// TIA Portal V18 program export: 1 tag tables, 3 data types, 16 data blocks, 44 code blocks (in call order from the OBs), 85 instance data blocks

VAR_GLOBAL   // PLC tag table "Default tag table"
   ESTOP_Button AT %I0.0 : Bool;   // Emergency button
   JOGNEG_BTN_Z1 AT %I0.2 : Bool;   // Z1 - Jogging Negative -> In order to execute this, real button sholud be pressed
   JOGPOS_BTN_Z1 AT %I0.1 : Bool;   // Z1 - Jogging Positive -> In order to execute this, real button sholud be pressed
   JOGNEG_BTN_Z2 AT %I0.4 : Bool;   // Z2 - Jogging Negative -> In order to execute this, real button sholud be pressed
   JOGPOS_BTN_Z2 AT %I0.3 : Bool;   // Z2 - Jogging Positive -> In order to execute this, real button sholud be pressed
   SENSOR_DOOR AT %I0.5 : Bool;   // Door Sensor Front
   Load_Cell_Ink AT %IW66 : UInt;
   Load_Cell_Waste AT %IW64 : UInt;
   SENSOR_DOOR_2 AT %I0.6 : Bool;   // Door Sensor Front
   UV_Error_Signal AT %I0.7 : Bool;   // Error signal from UV lamp, 0-4 V error, 16-24 V ok;
   SENSOR_DOOR_3 AT %I1.0 : Bool;   // Door Sensor Side
   SENSOR_DOOR_4 AT %I1.1 : Bool;   // Door Sensor Side
   SENSOR_DOOR_5 AT %I1.2 : Bool;   // Door Sensor Fluid Supply
   SENSOR_DOOR_6 AT %I1.3 : Bool;   // Door Sensor Fluid Supply
   TemperatureSensor AT %IW116 : UInt;
   CappingSensor AT %IW118 : UInt;
   AnalogInput3 AT %IW120 : UInt;
   AnalogInput4 AT %IW122 : UInt;
   "Roller Encoder" AT %ID1000 : DWord;
   "STO-B_Output" AT %Q0.0 : Bool;   // Safty Torque Off , for CMMO [Port X3, Pin ..]and CMMP in order to release a break
   Roller_Output AT %Q0.6 : Bool;
   Heater_Output AT %Q1.0 : Bool;   // Heater: ON/OFF_PLC/3.2B; %Q1.0
   LED_1_Output AT %Q0.4 : Bool;
   LED_2_Output AT %Q0.5 : Bool;
   Heater_PWM_pulseduration AT %QW1008 : Int;   // Heater: SETPOINT_PLC/3.2C; %Q0.3
   Capping_Station_PTO AT %Q0.1 : Bool;
   Capping_Station_DIR AT %Q0.2 : Bool;
   Roller_PWM_pulseduration AT %QW1014 : Int;
   UV_CTRL_ON_OFF AT %Q0.7 : Bool;
   UV_Dimming AT %QW106 : UInt;
   Stacklight01 AT %Q50.0 : Bool;
   Stacklight02 AT %Q50.1 : Bool;
   RollerDirection AT %Q1.1 : Bool;
   Tag_1 AT %IW1000 : Hw_Hsc;
END_VAR

TYPE "DT_FML_PRM_FILE"
   STRUCT
      Control : Int;
      BitSequenceNr : Int;
      Data : Array[1..6] of Byte;
   END_STRUCT;
END_TYPE

TYPE "DT_FML_REF"
   STRUCT
      InData : Struct
         FHPP : Array[1..16] of Byte;
         FPC : Array[1..8] of Byte;
         FHPPplus : Array[1..10] of DInt;
      END_STRUCT;
      OutData : Struct
         FHPP : Array[1..16] of Byte;
         FPC : Array[1..8] of Byte;
         FHPPplus : Array[1..10] of DInt;
      END_STRUCT;
      Modbus : Bool;
      DeviceType : String[16];
      MemberID : Int;
      MemberIDmax : Int;
      Done : Bool;
      Err : Bool;
      PNU : Word;
      ActPNU : Word;
      ReqID : Int;
      RespID : Int;
      FPCC_Modus : Byte;
      FPCS_Modus : Byte;
      FPCC_Packet : "DT_FML_PRM_FILE";
      FPCS_Packet : "DT_FML_PRM_FILE";
      Subindex : Byte;
      ActSubindex : Byte;
      DatatypeWR : Byte;
      DatatypeRD : Byte;
      ParamValueWR : DInt;
      ParamValueRD : DInt;
   END_STRUCT;
END_TYPE

TYPE "DT_FML_STATUS"
   STRUCT
      Err : Bool;
      Cat : Int;
      ID : DInt;
   END_STRUCT;
END_TYPE

DATA_BLOCK "Auxiliary_variables"   // DB17
{ S7_Optimized_Access := 'TRUE' }
VERSION : 0.1
   VAR
      GlobalEnableAxis : Bool;   // Variable enables Enable_machine [FC5]
      DisableAxis : Bool;   // Variable enables Stop_machine_sequence [FC4]
      StartFunction : Bool;   // Variable enables Function_sequence [FC6]
      ESTOP : Bool;   // Variable enables Emergancy_stop_sequence [FC3]
      ResetErrors : Bool;   // Variable enables Reset_error_sequence [FB14]
      Position_range_Z2 : DInt;   // Check if position is in the range Z2
      Mov_permission_Z2_Absolute : Bool;   // Permission to move Z2 (Input Axis_Mov Z2)
      Mov_permission_Z2_Relative : Bool;
      Stop_Z2_Out : Bool;   // Stop Z2 movement (Output for Axis_Mov Z2 block)
      Reset_command_Z2 : Bool;   // Reset Mov_mode / Mode_mode = 0 / Input for BOOL_DEMUX and Output for Axis_Mov Z2 Block
      Reset_error_jump_Z2 : Bool;   // Using in order to eliminate double write
      Position_range_X : DInt;   // Check if position is in the range X
      Mov_permission_X_Absolute : Bool;   // Permission to move Z2 (Input Axis_Mov X)
      Mov_permission_X_Relative : Bool;
      Stop_X_Out : Bool;   // Stop X movement (Output for Axis_Mov X block)
      Reset_command_X : Bool;   // Reset Mov_mode / Mode_mode = 0 / Input for BOOL_DEMUX and Output for Axis_Mov X Block
      Reset_error_jump_X : Bool;   // Using in order to eliminate double write
      Reset_command_Y : Bool;   // Reset Mov_mode / Mode_mode = 0 / Input for BOOL_DEMUX and Output for Axis_Mov Y Block
      Reset_error_jump_Y : Bool;   // Using in order to eliminate double write
      Stop_Y_Out : Bool;   // Stop Y movement (Output for Axis_Mov Y block)
      Mov_permission_Y_Absolute : Bool;   // Permission to move Y (Input Axis_Mov Y)
      Mov_permission_Y_Relative : Bool;
      Position_range_Y : DInt;   // Check if position is in the range Y
      Position_range_Z1 : DInt;   // Check if position is in the range Z1
      Mov_permission_Z1_Absolute : Bool;   // Permission to move Z1 (Input Axis_Mov Z1)
      Mov_permission_Z1_Relative : Bool;
      Stop_Z1_Out : Bool;   // Stop Z1 movement (Output for Axis_Mov Z1 block)
      Reset_command_Z1 : Bool;   // Reset Mov_mode / Mode_mode = 0 / Input for BOOL_DEMUX and Output for Axis_Mov Z1 Block
      Reset_error_jump_Z1 : Bool;   // Using in order to eliminate double write
      Stop_all_axis_command : Bool;   // Execute via Step6 ( in Main) / Stop all axis
      Mov_mode_reset_ALL_Axis : Bool;   // Reset Mov_mode after stopping all axis
      JogPosBTN_Z1_RisingEdge : Bool;   // Auxiliary variable used to execute JogPos Button
      JogNegBTN_Z1_RisingEdge : Bool;   // Auxiliary variable used to execute JogNeg Button
      JogPosBTN_Z1_FallingEdge : Bool;   // Auxiliary variable used to execute JogPos Button
      JogNegBTN_Z1_FallingEdge : Bool;   // Auxiliary variable used to execute JogNeg Button
      JogPosBTN_Z2_RisingEdge : Bool;   // Auxiliary variable used to execute JogPos Button
      JogNegBTN_Z2_RisingEdge : Bool;   // Auxiliary variable used to execute JogNeg Button
      JogPosBTN_Z2_FallingEdge : Bool;   // Auxiliary variable used to execute JogPos Button
      JogNegBTN_Z2_FallingEdge : Bool;   // Auxiliary variable used to execute JogNeg Button
      Heater_Start : Bool;   // Variable used to activate the heater during the spreading sequence
      PID_PWM_Output : Bool;   // PID Compact block -> Output
      CMD_Y_EM : Bool;
      CMD_X_EM : Bool;
      CMD_Z1_EM : Bool;
      CMD_Z2_EM : Bool;
      RelativeZ1 : Bool;
   END_VAR
BEGIN
END_DATA_BLOCK

DATA_BLOCK "ChaosDB"   // DB18
{ S7_Optimized_Access := 'TRUE' }
VERSION : 0.1
   VAR
      Step0 : Bool;
      Step1 : Bool;
      Step2 : Bool;
      Step3 : Bool;
      Step4 : Bool;
      Step5 : Bool;
      Step6 : Bool;
      Step7 : Bool;
      Step10 : Bool;
      Step20 : Bool;
      Step21 : Bool;
      Step1_Step2 : Bool;
      Step2_Step3 : Bool;
      Step2_Step5 : Bool;
      Step4_Step5 : Bool;
      Step2_Step20 : Bool;
      Step3_Step_4 : Bool;
      Step4_Step6 : Bool;
      Step4_Step10 : Bool;
      Step4_Step20 : Bool;
      Step5_Step2 : Bool;
      Step6_Step7 : Bool;
      Step7_Step4 : Bool;
      Step10_Step2 : Bool;
      Step20_Step21 : Bool;
      Step21_Step2 : Bool;
      Edge_Step1M : Bool;
      Edge_Step1S : Bool;
      Edge_Reset_Z2_M : Bool;
      Edge_Reset_Z2_S : Bool;
      Edge_Reset_X_S : Bool;
      Edge_Reset_X_M : Bool;
      Edge_Reset_Y_S : Bool;
      Edge_Reset_Y_M : Bool;
      Reset_error_main : Bool;
      Edge_M_res_err_main : Bool;
      Edge_S_res_err_main : Bool;
      Edge_Reset_Z1_S : Bool;
      Edge_Reset_Z1_M : Bool;
      Monitor_state : Bool;   // Auxiliary variable
      Edge_S_ResCMMOZ2 : Bool;   // Reset CMMO Z2 Controller
      Edge_M_ResCMMOZ2 : Bool;   // Reset CMMO Z2 Controller
      Restart_CMMO_Z2_Cmd : Bool;   // Reset CMMO Z2 Controller
      Edge_S_ResCMMOZ1 : Bool;   // Reset CMMO Z1Controller
      Edge_M_ResCMMOZ1 : Bool;   // Reset CMMO Z1 Controller
      Restart_CMMO_Z1_Cmd : Bool;   // Reset CMMO Z1Controller
      Edge_S_ResCMMPX : Bool;   // Reset CMMP X Controller
      Edge_M_ResCMMPX : Bool;   // Reset CMMP X Controller
      Restart_CMMP_X_Cmd : Bool;   // Reset CMMP X Controller
      Edge_S_ResCMMPY : Bool;   // Reset CMMP Y Controller
      Edge_M_ResCMMPY : Bool;   // Reset CMMP Y Controller
      Restart_CMMP_Y_Cmd : Bool;   // Reset CMMP Y Controller
      Z2_Stop_E : Bool;
      Z2_Stop_EM : Bool;
   END_VAR
BEGIN
END_DATA_BLOCK

DATA_BLOCK "DevTestBlock"   // DB47
{ S7_Optimized_Access := 'FALSE' }
VERSION : 0.1
   VAR
      EnableAxisTest : Bool;
      Z2Halt : Bool;
      Z1Halt : Bool;
      XHalt : Bool;
      YHalt : Bool;
      GlobalHalt : Bool;
      TaskZ2E : Bool;
      TaskZ1M : Bool;
      TaskZ2M : Bool;
      TaskXM : Bool;
      TaskYM : Bool;
      TestResetCommand : Bool;
      TestResetZ1 : Bool;
      TestResetZ2 : Bool;
      TestResetX : Bool;
      TestResetY : Bool;
      DoorSensor : Bool := true;   // True for testing to disable door sensors
      "Weight Test value" : UInt;
      DoorSensorPrintboxSkip : Bool := true;
      DoorSensor_Side : Bool := false;
      DoorSensor_PrintBox : Bool;
      AXIS_ackerror : Bool;
      AXIS_X_enable : Bool;
      AXIS_Y_enable : Bool;
      AXIS_Z1_enable : Bool;
      AXIS_jog1 : Bool := false;
      AXIS_jog2 : Bool;
      AXIS_X_velocity : Real;
      AXIS_X_position : Int;
      AXIS_execute : Bool;
      ConfigEPos : DWord := 16#0000_000F;
      "AXIS Warning" : Bool := false;
      "AXIS Error Fault" : Bool := false;
      "AXIS Enabled" : Bool := false;
      "AXIS Ready" : Bool := false;
      PurgeX : DInt := 480000;
      PurgeY : DInt := 90000;
      PurgeVelocity : DInt := 300;
      PurgeMove : Bool;
      "OLD off" : Bool;
      LED1 : Bool;
      LED2 : Bool;
      CappingHoming : Bool;
      reset : Bool;
      DamagedDoorSensorTemp : Bool := false;
      CappingEnable : Bool;
      TestYvelocity : DInt := 100000;
      TestingCappingStation : Bool;
      TestCapping01 : Bool;
      TestCapping02 : Bool;
      TestCapping03 : Bool;
      TestCappingNotUsed : Bool;
      ResetCounters : Bool;
      RET_VAL : Int;
      WebServerTest : Int := 1;
   END_VAR
BEGIN
END_DATA_BLOCK

DATA_BLOCK "MachineDB"   // DB22
{ S7_Optimized_Access := 'FALSE' }
VERSION : 0.1
   VAR RETAIN
      SerialNumber : Int := 2011;
      AutomateVersion : Int := 6;
      MachineType : String := 'ArmadilloV7BR';   // Not writable from HMI
      MachineLimit : Struct
         XSafety : Struct
            PosMax : DInt := 0;
            PosMin : DInt := 0;
            SafetyMargin : DInt;
            VelocityMax : DInt;
            VelocityMin : DInt;
         END_STRUCT;
         YSafety : Struct
            PosMax : DInt := 0;
            PosMin : DInt := 0;
            SafetyMargin : DInt;
            VelocityMax : DInt;
            VelocityMin : DInt;
         END_STRUCT;
         Z1Safety : Struct
            PosMax : DInt := 0;
            PosMin : DInt := 0;
            SafetyMargin : DInt;
            VelocityMax : DInt;
            VelocityMin : DInt;
         END_STRUCT;
         Z2Safety : Struct
            PosMax : DInt := 0;
            PosMin : DInt := 0;
            SafetyMargin : DInt;
            VelocityMax : DInt;
            VelocityMin : DInt;
         END_STRUCT;
         Heater : Struct
            FeedboxStart : DInt;
            FeedboxEnd : DInt;
            PrintboxStart : DInt;
            PrintboxEnd : DInt;
         END_STRUCT;
      END_STRUCT;
      ArmadilloOption : Struct
         MachineTypeNext : String := 'ArmadilloV7BR';
         DoorOption : Int := 3;   // SAFETY OPTION, ASK BEFORE CHANGING
         DoorOptionNext : Int := 3;
         DepowderingBox : Int;   // 0 if no box; 1 is we use V1 of the box;
         DepowderingBoxNext : Int;   // 0 if no box; 1 is we use V1 of the box;
         ZAxisDriveOption : String := 'CMMT';   // CMMT;CMMS;
         ZAxisDriveOptionNext : String := 'CMMT';   // CMMT;CMMS;
         UVOption : Int := 1;   // 0 means no UV lamp; 1 version of the UV lamp;
         UVOptionNext : Int := 1;   // 0 means no UV lamp; 1 version of the UV lamp;
         StacklightOption : Int := 1;   // 0 means no Stacklight; 1 version of the Stacklight;
         StacklightOptionNext : Int := 1;   // 0 means no Stacklight; 1 version of the Stacklight;
         CappingStationOption : Int := 1;   // 0 means no Capping Station; 1 version of the Capping Station;
         CappingStationOptionNext : Int := 1;   // 0 means no Capping Station; 1 version of the Capping Station;
      END_STRUCT;
      MachineLimitSecondary : Struct
         NoGoZone01 : Struct   // Temporary not used -> go to DepowderingBoxDimensions
            NoGoZone01_Xstart : DInt;   // Start of the No Go Zone for Depowdering Box
            NoGoZone01_Xend : DInt;   // Start of the No Go Zone for Depowdering Box
            NoGoZone01_Ystart : DInt;   // Start of the No Go Zone for Depowdering Box
            NoGoZone01_Yend : DInt;   // End of the No Go Zone for Depowdering Box
            NoGoZone01_Z1start : DInt;   // Start of the No Go Zone for Depowdering Box
            NoGoZone01_Z1end : DInt;   // End of the No Go Zone for Depowdering Box
            NoGoZone01_Z2start : DInt;   // Start of the No Go Zone for Depowdering Box
            NoGoZone01_Z2end : DInt;   // End of the No Go Zone for Depowdering Box
         END_STRUCT;
      END_STRUCT;
      MachineTypeString : Struct
         _sArmadilloDev : String := 'ArmadilloDev';   // Not writable from HMI
         _sArmadilloV2 : String := 'ArmadilloV2';   // Not writable from HMI
         _sArmadilloBRV2 : String := 'ArmadilloBRV2';   // Not writable from HMI
         _sArmadilloXLV2 : String := 'ArmadilloXLV2';   // Not writable from HMI
         _sArmadilloXLBRV2 : String := 'ArmadilloXLBRV2';   // Not writable from HMI
         _sArmadilloV6 : String := 'ArmadilloV6';   // Machine 2007;
         _sArmadilloV6BR : String := 'ArmadilloV6BR';   // Machine 2007;
         _sArmadilloV7 : String := 'ArmadilloV7';   // Machine 2009; 2011;
         _sArmadilloV7BR : String := 'ArmadilloV7BR';   // Machine 2009; 2011;
         _sArmadilloXLV7 : String := 'ArmadilloXLV7';   // Machine 2010;
         _sArmadilloXLV7BR : String := 'ArmadilloXLV7BR';   // Machine 2010;
      END_STRUCT;
      ArmadilloDevMachine : Struct   // Software limit for the Armadillo Dev machine
         XSafety : Struct
            PosMax : DInt := 454000;
            PosMin : DInt := -3000;
            SafetyMargin : DInt := 0;
            VelocityMax : DInt := 500;
            VelocityMin : DInt := 0;
         END_STRUCT;
         YSafety : Struct
            PosMax : DInt := 1100000;
            PosMin : DInt := -3000;
            SafetyMargin : DInt := 0;
            VelocityMax : DInt := 500;
            VelocityMin : DInt;
         END_STRUCT;
         Z1Safety : Struct
            PosMax : DInt := 297850;
            PosMin : DInt := -3000;
            SafetyMargin : DInt := 0;
            VelocityMax : DInt := 20;
            VelocityMin : DInt;
         END_STRUCT;
         Z2Safety : Struct
            PosMax : DInt := 297850;
            PosMin : DInt := -3000;
            SafetyMargin : DInt := 0;
            VelocityMax : DInt := 20;
            VelocityMin : DInt;
         END_STRUCT;
         Heater : Struct
            FeedboxStart : DInt := 100000;
            FeedboxEnd : DInt := 400000;
            PrintboxStart : DInt := 300000;
            PrintboxEnd : DInt := 765000;
         END_STRUCT;
      END_STRUCT;
      ArmadilloBRMachine : Struct   // Software limit for the Armadillo Dev machine
         XSafety : Struct
            PosMax : DInt := 454000;
            PosMin : DInt := -3000;
            SafetyMargin : DInt;
            VelocityMax : DInt;
            VelocityMin : DInt;
         END_STRUCT;
         YSafety : Struct
            PosMax : DInt := 1100000;
            PosMin : DInt := -3000;
            SafetyMargin : DInt;
            VelocityMax : DInt;
            VelocityMin : DInt;
         END_STRUCT;
         Z1Safety : Struct
            PosMax : DInt := 94000;   // v1 = 210500
            PosMin : DInt := -3000;
            SafetyMargin : DInt;
            VelocityMax : DInt;
            VelocityMin : DInt;
         END_STRUCT;
         Z2Safety : Struct
            PosMax : DInt := 94000;   // v1 = 210500
            PosMin : DInt := -3000;
            SafetyMargin : DInt;
            VelocityMax : DInt;
            VelocityMin : DInt;
         END_STRUCT;
         Heater : Struct
            FeedboxStart : DInt;
            FeedboxEnd : DInt;
            PrintboxStart : DInt;
            PrintboxEnd : DInt;
         END_STRUCT;
      END_STRUCT;
      ArmadilloXLMachine : Struct   // Software limit for the Armadillo Production machine
         XSafety : Struct
            PosMax : DInt := 516000;
            PosMin : DInt := -3000;
            SafetyMargin : DInt;
            VelocityMax : DInt;
            VelocityMin : DInt;
         END_STRUCT;
         YSafety : Struct
            PosMax : DInt := 1380000;
            PosMin : DInt := -3000;
            SafetyMargin : DInt;
            VelocityMax : DInt;
            VelocityMin : DInt;
         END_STRUCT;
         Z1Safety : Struct
            PosMax : DInt := 302000;
            PosMin : DInt := -500;
            SafetyMargin : DInt;
            VelocityMax : DInt;
            VelocityMin : DInt;
         END_STRUCT;
         Z2Safety : Struct
            PosMax : DInt := 302000;
            PosMin : DInt := -500;
            SafetyMargin : DInt;
            VelocityMax : DInt;
            VelocityMin : DInt;
         END_STRUCT;
         Heater : Struct
            FeedboxStart : DInt;
            FeedboxEnd : DInt;
            PrintboxStart : DInt;
            PrintboxEnd : DInt;
         END_STRUCT;
      END_STRUCT;
      ArmadilloXLBRMachine : Struct   // Software limit for the Armadillo Production machine
         XSafety : Struct
            PosMax : DInt := 516000;
            PosMin : DInt := -3000;
            SafetyMargin : DInt;
            VelocityMax : DInt;
            VelocityMin : DInt;
         END_STRUCT;
         YSafety : Struct
            PosMax : DInt := 1380000;
            PosMin : DInt := -3000;
            SafetyMargin : DInt;
            VelocityMax : DInt;
            VelocityMin : DInt;
         END_STRUCT;
         Z1Safety : Struct
            PosMax : DInt := 210500;
            PosMin : DInt := -3000;
            SafetyMargin : DInt;
            VelocityMax : DInt;
            VelocityMin : DInt;
         END_STRUCT;
         Z2Safety : Struct
            PosMax : DInt := 210500;
            PosMin : DInt := -3000;
            SafetyMargin : DInt;
            VelocityMax : DInt;
            VelocityMin : DInt;
         END_STRUCT;
         Heater : Struct
            FeedboxStart : DInt;
            FeedboxEnd : DInt;
            PrintboxStart : DInt;
            PrintboxEnd : DInt;
         END_STRUCT;
      END_STRUCT;
      ArmadilloV6Machine : Struct   // 2007 Eurostar Software limit for the Armadillo V6 machine
         XSafety : Struct
            PosMax : DInt := 500000;
            PosMin : DInt := 0;
            SafetyMargin : DInt := 5000;
            VelocityMax : DInt := 500;
            VelocityMin : DInt := 0;
         END_STRUCT;
         YSafety : Struct
            PosMax : DInt := 1365000;
            PosMin : DInt := 0;
            SafetyMargin : DInt := 5000;
            VelocityMax : DInt := 500;
            VelocityMin : DInt;
         END_STRUCT;
         Z1Safety : Struct
            PosMax : DInt := 300000;
            PosMin : DInt := 0;
            SafetyMargin : DInt := 2000;
            VelocityMax : DInt;
            VelocityMin : DInt;
         END_STRUCT;
         Z2Safety : Struct
            PosMax : DInt := 300000;
            PosMin : DInt := 0;
            SafetyMargin : DInt := 2000;
            VelocityMax : DInt;
            VelocityMin : DInt;
         END_STRUCT;
         Heater : Struct
            FeedboxStart : DInt := 270000;
            FeedboxEnd : DInt := 580000;
            PrintboxStart : DInt := 580000;
            PrintboxEnd : DInt := 880000;
         END_STRUCT;
      END_STRUCT;
      ArmadilloV6BRMachine : Struct   // 2007 Eurostar Software limit for the Armadillo V6 Bed Reduction machine
         XSafety : Struct
            PosMax : DInt := 500000;
            PosMin : DInt := 0;
            SafetyMargin : DInt := 5000;
            VelocityMax : DInt := 500;
            VelocityMin : DInt;
         END_STRUCT;
         YSafety : Struct
            PosMax : DInt := 1365000;
            PosMin : DInt := 0;
            SafetyMargin : DInt := 5000;
            VelocityMax : DInt := 500;
            VelocityMin : DInt;
         END_STRUCT;
         Z1Safety : Struct
            PosMax : DInt := 90000;   // v1 = 210500
            PosMin : DInt := 0;
            SafetyMargin : DInt := 2000;
            VelocityMax : DInt;
            VelocityMin : DInt;
         END_STRUCT;
         Z2Safety : Struct
            PosMax : DInt := 90000;   // v1 = 210500
            PosMin : DInt := 0;
            SafetyMargin : DInt := 2000;
            VelocityMax : DInt;
            VelocityMin : DInt;
         END_STRUCT;
         Heater : Struct
            FeedboxStart : DInt := 470000;
            FeedboxEnd : DInt := 580000;
            PrintboxStart : DInt := 580000;
            PrintboxEnd : DInt := 680000;
         END_STRUCT;
      END_STRUCT;
      ArmadilloV7Machine : Struct   // 2009, 2011 Normal Software limit for the Armadillo V6 machine
         XSafety : Struct
            PosMax : DInt := 435000;
            PosMin : DInt := -3000;
            SafetyMargin : DInt := 5000;
            VelocityMax : DInt := 500;
            VelocityMin : DInt := 0;
         END_STRUCT;
         YSafety : Struct
            PosMax : DInt := 1065000;
            PosMin : DInt := -3000;
            SafetyMargin : DInt := 5000;
            VelocityMax : DInt := 500;
            VelocityMin : DInt;
         END_STRUCT;
         Z1Safety : Struct
            PosMax : DInt := 312000;
            PosMin : DInt := 0;
            SafetyMargin : DInt := 2000;
            VelocityMax : DInt;
            VelocityMin : DInt;
         END_STRUCT;
         Z2Safety : Struct
            PosMax : DInt := 312000;
            PosMin : DInt := 0;
            SafetyMargin : DInt := 2000;
            VelocityMax : DInt;
            VelocityMin : DInt;
         END_STRUCT;
         Heater : Struct
            FeedboxStart : DInt := 100000;
            FeedboxEnd : DInt := 430000;
            PrintboxStart : DInt := 430000;
            PrintboxEnd : DInt := 740000;
         END_STRUCT;
      END_STRUCT;
      ArmadilloV7BRMachine : Struct   // 2009, 2011 Normal Software limit for the Armadillo V6 Bed Reduction machine
         XSafety : Struct
            PosMax : DInt := 435000;
            PosMin : DInt := -3000;
            SafetyMargin : DInt := 5000;
            VelocityMax : DInt := 500;
            VelocityMin : DInt;
         END_STRUCT;
         YSafety : Struct
            PosMax : DInt := 1065000;
            PosMin : DInt := -3000;
            SafetyMargin : DInt := 5000;
            VelocityMax : DInt := 500;
            VelocityMin : DInt;
         END_STRUCT;
         Z1Safety : Struct
            PosMax : DInt := 86000;
            PosMin : DInt := 0;
            SafetyMargin : DInt := 2000;
            VelocityMax : DInt;
            VelocityMin : DInt;
         END_STRUCT;
         Z2Safety : Struct
            PosMax : DInt := 86000;
            PosMin : DInt := 0;
            SafetyMargin : DInt := 2000;
            VelocityMax : DInt;
            VelocityMin : DInt;
         END_STRUCT;
         Heater : Struct
            FeedboxStart : DInt := 250000;
            FeedboxEnd : DInt := 360000;
            PrintboxStart : DInt := 360000;
            PrintboxEnd : DInt := 490000;
         END_STRUCT;
      END_STRUCT;
      ArmadilloXLV7Machine : Struct   // 2010 XL Software limit for the Armadillo V6 machine
         XSafety : Struct
            PosMax : DInt := 500000;
            PosMin : DInt := -3000;
            SafetyMargin : DInt := 5000;
            VelocityMax : DInt := 500;
            VelocityMin : DInt := 0;
         END_STRUCT;
         YSafety : Struct
            PosMax : DInt := 1365000;
            PosMin : DInt := -3000;
            SafetyMargin : DInt := 5000;
            VelocityMax : DInt := 500;
            VelocityMin : DInt;
         END_STRUCT;
         Z1Safety : Struct
            PosMax : DInt := 312000;
            PosMin : DInt := 0;
            SafetyMargin : DInt := 2000;
            VelocityMax : DInt;
            VelocityMin : DInt;
         END_STRUCT;
         Z2Safety : Struct
            PosMax : DInt := 312000;
            PosMin : DInt := 0;
            SafetyMargin : DInt := 2000;
            VelocityMax : DInt;
            VelocityMin : DInt;
         END_STRUCT;
         Heater : Struct
            FeedboxStart : DInt := 150000;
            FeedboxEnd : DInt := 610000;
            PrintboxStart : DInt := 610000;
            PrintboxEnd : DInt := 1100000;
         END_STRUCT;
      END_STRUCT;
      ArmadilloXLV7BRMachine : Struct   // 2010 XL Software limit for the Armadillo V6 Bed Reduction machine
         XSafety : Struct
            PosMax : DInt := 500000;
            PosMin : DInt := -3000;
            SafetyMargin : DInt := 5000;
            VelocityMax : DInt := 500;
            VelocityMin : DInt;
         END_STRUCT;
         YSafety : Struct
            PosMax : DInt := 1365000;
            PosMin : DInt := -3000;
            SafetyMargin : DInt := 5000;
            VelocityMax : DInt := 500;
            VelocityMin : DInt;
         END_STRUCT;
         Z1Safety : Struct
            PosMax : DInt := 86000;
            PosMin : DInt := 0;
            SafetyMargin : DInt := 2000;
            VelocityMax : DInt;
            VelocityMin : DInt;
         END_STRUCT;
         Z2Safety : Struct
            PosMax : DInt := 86000;
            PosMin : DInt := 0;
            SafetyMargin : DInt := 2000;
            VelocityMax : DInt;
            VelocityMin : DInt;
         END_STRUCT;
         Heater : Struct
            FeedboxStart : DInt := 440000;
            FeedboxEnd : DInt := 620000;
            PrintboxStart : DInt := 620000;
            PrintboxEnd : DInt := 770000;
         END_STRUCT;
      END_STRUCT;
      DepowderingBoxDimensions : Struct   // Should be integrated with machine limits in the future
         DepowderingBoxHeight : DInt := 27000;
         DepowderingBoxWidth : DInt := 0;
         DepowderingBoxMargin : DInt := 3000;
         DepowderingBoxNormal : Struct
            DepowderingBoxNormalXstart : DInt := 0;
            DepowderingBoxNormalXend : DInt := 550000;
            DepowderingBoxNormalYstart : DInt := 180000;
            DepowderingBoxNormalYend : DInt := 1500000;
         END_STRUCT;
         DepowderingBoxXL : Struct
            DepowderingBoxXLXstart : DInt := 0;
            DepowderingBoxXLXend : DInt := 550000;
            DepowderingBoxXLYstart : DInt := 190000;
            DepowderingBoxXLYend : DInt := 1500000;
         END_STRUCT;
      END_STRUCT;
   END_VAR
BEGIN
END_DATA_BLOCK

DATA_BLOCK "MainDB"   // DB30
{ S7_Optimized_Access := 'TRUE' }
VERSION : 0.1
   VAR
      Monitor : Bool;
      Step0M : Bool;
      Step0 : Bool;
      Step10 : Bool;
      Step20 : Bool;
      Step30 : Bool;
      Step40 : Bool;
      Step50 : Bool;
      Step0_10 : Bool;
      Step10_20 : Bool;
      Step20_30 : Bool;
      Step30_40 : Bool;
      Step40_50 : Bool;
      Step50_10 : Bool;
      ESTOPEdgeMemory : Bool;
      ESTOPEdge : Bool;
      AllAxisFaultRelease : Bool;
      Step0MConfig : Bool;
   END_VAR
BEGIN
END_DATA_BLOCK

DATA_BLOCK "WebDB"   // DB5
{ S7_Optimized_Access := 'FALSE' }
VERSION : 0.1
   VAR
      Enabled_Devices : Bool;   // Diagnostic value, necessary in step 3 (Check if system is ready); TRUE if OK;
      Ready_Devices : Bool;   // Diagnostic value, necessary in step 3 (Check if system is ready); TRUE if OK;
      Warning_Devices : Bool;   // Diagnostic value, necessary in step 3 (Check if system is ready); TRUE if OK;
      Fault_Devices : Bool;   // Diagnostic value, necessary in step 3 (Check if system is ready); TRUE if OK;
      diagMode : UInt := 1;   // Diagnostic mode : 0
      myLADDR : HW_ANY := 52;   // ID of CPUExecutUnit : 52 PLC ID: 64
      returnValue : Int;   // No error: 0
      CountDiagDetails : UInt;   // Should always be 0
      PLCDiag : DIS;   // Read value of diagnostic
      Start_Machine : Bool;   // Button - Start Machine
      Stop_Machine : Bool;   // Button - Stop Machine
      Reset_error : Bool;   // Button - Reset error after emergancy stop and other situation
      Stop_All_Axis : Bool;
      XInput : Struct
         EnableDrive : Bool;
         Stop : Bool;
         Halt : Bool;
         Brake : Bool;
         ResetFault : Bool;
         HMIAccessLocked : Bool;
         OPM : Int;   // Operating Mode ???
         StartTask : Bool;
         StartHoming : Bool;
         JogPos : Bool;
         JogNeg : Bool;
         TeachActValue : Bool;
         ClearRemPos : Bool;
         Relative : Bool;
         DeactivateStrokeLimit : Bool;
         ExecuteFunction : Bool;
         RecordNo : Int;
         SetFunctionNumber : Int;
         SetFunctionGroup : Int;
         SetValueVelocity : DInt := 20;
         SetValuePosition : DInt;
         SetValueForceRamp : DInt;
         SetValueForce : DInt;
         SetValueRotRamp : DInt;
         SetValueRotSpeed : DInt;
      END_STRUCT;
      XOutput : Struct
         DriveEnabled : Bool;
         Ready : Bool;
         Warning : Bool;
         Fault : Bool;
         SupplyVoltPresent : Bool;
         ControlFCT_HMI : Bool;
         StateOPM : Int;
         HaltNotActive : Bool;
         AckStart : Bool;
         MC : Bool;
         AckTeach : Bool;
         DriveMoving : Bool;
         DragError : Bool;
         StandStillControl : Bool;
         HomingValid : Bool;
         ActualRecordNo : Int;
         RC1 : Bool;
         RCC : Bool;
         VelocityLimitReached : Bool;
         StrokeLimitReached : Bool;
         FunctionIsActive : Bool;
         ActualFunctionNumber : Int;
         ActualFunctionGroup : Int;
         ActualPosition : DInt;
         ActualVelocity : DInt;
         ActualForce : DInt;
         ActualRotRamp : DInt;
         ActualRotSpeed : DInt;
      END_STRUCT;
      XAddOn1 : Struct
         XTargetRange : DInt := 1000;
         XTargetReached : Bool;
         XOverrange : Bool;
         Error_message_X : DInt;   // Number of error in DINT. Check error in CMMP documentation
         Restart_CMMO_X : Bool;   // Restart CMMP X controller
      END_STRUCT;
      YInput : Struct
         EnableDrive : Bool;
         Stop : Bool;
         Halt : Bool;
         Brake : Bool;
         ResetFault : Bool;
         HMIAccessLocked : Bool;
         OPM : Int;   // Operating Mode ???
         StartTask : Bool;
         StartHoming : Bool;
         JogPos : Bool;
         JogNeg : Bool;
         TeachActValue : Bool;
         ClearRemPos : Bool;
         Relative : Bool;
         DeactivateStrokeLimit : Bool;
         ExecuteFunction : Bool;
         RecordNo : Int;
         SetFunctionNumber : Int;
         SetFunctionGroup : Int;
         SetValueVelocity : DInt := 20;
         SetValuePosition : DInt;
         SetValueForceRamp : DInt;
         SetValueForce : DInt;
         SetValueRotRamp : DInt;
         SetValueRotSpeed : DInt;
      END_STRUCT;
      YOutput : Struct
         DriveEnabled : Bool;
         Ready : Bool;
         Warning : Bool;
         Fault : Bool;
         SupplyVoltPresent : Bool;
         ControlFCT_HMI : Bool;
         StateOPM : Int;
         HaltNotActive : Bool;
         AckStart : Bool;
         MC : Bool;
         AckTeach : Bool;
         DriveMoving : Bool;
         DragError : Bool;
         StandStillControl : Bool;
         HomingValid : Bool;
         ActualRecordNo : Int;
         RC1 : Bool;
         RCC : Bool;
         VelocityLimitReached : Bool;
         StrokeLimitReached : Bool;
         FunctionIsActive : Bool;
         ActualFunctionNumber : Int;
         ActualFunctionGroup : Int;
         ActualPosition : DInt;
         ActualVelocity : DInt;
         ActualForce : DInt;
         ActualRotRamp : DInt;
         ActualRotSpeed : DInt;
      END_STRUCT;
      YAddOn1 : Struct
         YTargetRange : DInt := 1000;
         YTargetReached : Bool;
         YOverrange : Bool;
         Error_message_Y : DInt;   // Number of error in DINT. Check error in CMMP documentation
         Restart_CMMO_Y : Bool;   // Restart CMMP Y controller
      END_STRUCT;
      Z1Input : Struct
         EnableDrive : Bool;
         Stop : Bool;
         Halt : Bool;
         Brake : Bool;
         ResetFault : Bool;
         HMIAccessLocked : Bool;
         OPM : Int;   // Operating Mode ???
         StartTask : Bool;
         StartHoming : Bool;
         JogPos : Bool;
         JogNeg : Bool;
         TeachActValue : Bool;
         ClearRemPos : Bool;
         Relative : Bool;
         DeactivateStrokeLimit : Bool;
         ExecuteFunction : Bool;
         RecordNo : Int;
         SetFunctionNumber : Int;
         SetFunctionGroup : Int;
         SetValueVelocity : DInt := 20;
         SetValuePosition : DInt;
         SetValueForceRamp : DInt;
         SetValueForce : DInt;
         SetValueRotRamp : DInt;
         SetValueRotSpeed : DInt;
      END_STRUCT;
      Z1Output : Struct
         DriveEnabled : Bool;
         Ready : Bool;
         Warning : Bool;
         Fault : Bool;
         SupplyVoltPresent : Bool;
         ControlFCT_HMI : Bool;
         StateOPM : Int;
         HaltNotActive : Bool;
         AckStart : Bool;
         MC : Bool;
         AckTeach : Bool;
         DriveMoving : Bool;
         DragError : Bool;
         StandStillControl : Bool;
         HomingValid : Bool;
         ActualRecordNo : Int;
         RC1 : Bool;
         RCC : Bool;
         VelocityLimitReached : Bool;
         StrokeLimitReached : Bool;
         FunctionIsActive : Bool;
         ActualFunctionNumber : Int;
         ActualFunctionGroup : Int;
         ActualPosition : DInt;
         ActualVelocity : DInt;
         ActualForce : DInt;
         ActualRotRamp : DInt;
         ActualRotSpeed : DInt;
      END_STRUCT;
      Z1AddOn1 : Struct
         Z1TargetRange : DInt := 1000;
         Z1TargetReached : Bool;
         Z1Overrange : Bool;
         Error_message_Z1 : DInt;   // Number of error in DINT. Check error in CMMO documentation
         Restart_CMMO_Z1 : Bool;   // Restart CMMO Z1 controller
      END_STRUCT;
      Z2Input : Struct
         EnableDrive : Bool;
         Stop : Bool;
         Halt : Bool;
         Brake : Bool;
         ResetFault : Bool;
         HMIAccessLocked : Bool;
         OPM : Int;   // Operating Mode ???
         StartTask : Bool;
         StartHoming : Bool;
         JogPos : Bool;
         JogNeg : Bool;
         TeachActValue : Bool;
         ClearRemPos : Bool;
         Relative : Bool;
         DeactivateStrokeLimit : Bool;
         ExecuteFunction : Bool;
         RecordNo : Int;
         SetFunctionNumber : Int;
         SetFunctionGroup : Int;
         SetValueVelocity : DInt := 20;
         SetValuePosition : DInt;
         SetValueForceRamp : DInt;
         SetValueForce : DInt;
         SetValueRotRamp : DInt;
         SetValueRotSpeed : DInt;
      END_STRUCT;
      Z2Output : Struct
         DriveEnabled : Bool;
         Ready : Bool;
         Warning : Bool;
         Fault : Bool;
         SupplyVoltPresent : Bool;
         ControlFCT_HMI : Bool;
         StateOPM : Int;
         HaltNotActive : Bool;
         AckStart : Bool;
         MC : Bool;
         AckTeach : Bool;
         DriveMoving : Bool;
         DragError : Bool;
         StandStillControl : Bool;
         HomingValid : Bool;
         ActualRecordNo : Int;
         RC1 : Bool;
         RCC : Bool;
         VelocityLimitReached : Bool;
         StrokeLimitReached : Bool;
         FunctionIsActive : Bool;
         ActualFunctionNumber : Int;
         ActualFunctionGroup : Int;
         ActualPosition : DInt;
         ActualVelocity : DInt;
         ActualForce : DInt;
         ActualRotRamp : DInt;
         ActualRotSpeed : DInt;
      END_STRUCT;
      Z2AddOn1 : Struct
         Z2TargetRange : DInt := 1000;
         Z2TargetReached : Bool;
         Z2Overrange : Bool;
         Error_message_Z2 : DInt;   // Number of error in DINT, Check error in CMMO documentation
         Restart_CMMO_Z2 : Bool;   // Restart CMMO Z2 controller
      END_STRUCT;
      Start_Roller : Bool;   // Set ON the rotations of the roller
      Stop_Roller : Bool;   // Reset OFF the rotations of the roller
      Output_Roller : Bool;
      SpreadParam : Struct
         spreadCycleYFirstPos : DInt;
         spreadCycleYSecondPos : DInt := 400000;
         spreadCycleYLastPos : DInt := 900000;
         Spread_BUSY : Bool;   // When spreading cycle is being executed - > TRUE
         Spread_DONE : Bool;   // Rising edge / When spreading cycle is done
         Spread_speed : DInt := 10;   // Value of speed (Y- axis) when the roller is above the printing bed
         Amount_of_layer : Int := 1;   // How many times do you want execute the spreading cycle ? How many powder layers do you want to spread ? Set value here.
         Spread_powder_stop : Bool;   // Spreading cycle - stop
         Spread_powder_execute : Bool;   // Spreading cycle - start / Don't forget set "Move_Feed" and "Move_Printing"
         Spread_Step_Z1 : DInt := 330;   // Relative movement / Set value / How much you want to up ?
         Spread_Step_Z2 : DInt := -300;   // Relative movement / How much you want to down ?
      END_STRUCT;
      Homing_all_axis : Bool;   // Press if you want execute homing for all axis
      SystemStatus : Struct   // System status: door sensor and emergency
         Emergency : Bool;   // Emergency button is active
         DoorSensor : Bool;
      END_STRUCT;
      Heater_ON : Bool;   // If you want to use the heater -> TRUE, if you don't want -> FALSE, Heater is activated during the spreading cycle
      PID_Heater_ON : Bool;   // If you want to use PID controller to control the temperature of powder - > TRUE , If the heater should be ON continuously -> FALSE, this option can be only activated when "Heater_ON" is TRUE
      WeightFluidTank : UInt;   // Weight in Kg
      WeightWastTank : UInt;   // Weight in Kg
      Heater_Setpoint : Real;   // Heating Setpoint [%] - future -> [Celsius]
      Heater_Sensor : Real;
      Heater_PDL : Real := 100.0;   // Pulse Duration Limit [%] - future -> [Celsius] set by technician or engineer in charge, don't change
      CappingStationInput : Struct
         CSMoveUP : Bool;   // Move capping station to the top position
         CSMoveDOWN : Bool;   // Move capping station to the bottom
      END_STRUCT;
      CappingStationOuput : Struct
         CSPositionUP : Bool;   // Confirmation of the top position reached
         CSPositionDOWN : Bool;   // Confirmation of the bottom position reached
         CSPosition : UInt;   // Actual position reading based on an estimation
         CSXYMotionLock : Bool;   // Motion lock to prevent destroying mechanism with the moving parts
      END_STRUCT;
      RollerAdjustableInput : Struct
         Mode : Int;   // 0; 1; 2; 3;
         SetSpeed : Real;   // %
         Direction : Bool;   // CW; CCW;
         OffsetSpeed : DInt;   // In mm/s
      END_STRUCT;
      RollerAdjustableOutput : Struct
         RollerDirection : Bool;
         RollerLinearVelocity : DInt;   // Relative speed of the roller surface in relation to the printbed surface
         setpointRPM : Real;
         RollerSpeedRPM : Real;   // Roller RPM - Measured
      END_STRUCT;
      UVLampInput : Struct   // Control of the UV lamp from NOAH
         UVLampEnable : Bool;   // Enable control block
         UVLampMode : Int;   // Choose lamp mode
         UVLampONOFF : Bool;   // Turn UV lamp ON and OFF
         UVLampSetpoint : Real;   // To enable the lamp, minimum 1V output
         UVLampMaintenance : Int;   // Maintenance mode to skip some of the safety rules
      END_STRUCT;
      UVLampOutput : Struct   // Status of the UV lamp in the PLC
         UVLampEnabled : Bool;
         UVLampWorking : Bool;   // 1 if lamp is ON; 0 if lamp is OFF
         UVLampError : Bool;   // 1 if OK; 0 if ERROR;
         UVLampIntensity : Real;   // Control Voltage 0-10V;
         UVLampStatus : Int;   // N/A
      END_STRUCT;
      StacklightInput : Struct   // Control of the Stacklight from NOAH
         StacklightEnable : Bool;   // 0 - working; 1 OFF;
         StacklightMode : Int;   // 0 - default mode;
         NOAHColor : Int;   // 0 red; 1 yellow; 2 green
         NOAHConnected : Bool;   // Checking if the connection is working
         NOAHPrinting : Bool;   // For the next version
         NOAHPaused : Bool;   // For the next version
         NOAHFluidError : Bool;
         StacklightMaintenance : Int;   // For special comands from NOAH
      END_STRUCT;
      StacklightOutput : Struct   // Status of the Stacklight in the PLC
         StacklightStatus : Int;   // N/A
         StaklightError : Bool;   // N/A
         StacklightColor : Int;   // 0 red; 1 yellow; 2 green
         StacklightCTRL01 : Bool;   // 0 Red; 1 Orange or Green;
         StacklightCTRL02 : Bool;   // 0 Orange; 1 Green;
      END_STRUCT;
      NoGoZone01AxisControl : Struct   // Control of the NoGoZone with restricted access
         NoGoMotionLockXmove : Bool;
         NoGoMotionLockXjog : Bool;
         NoGoMotionLockYmove : Bool;
         NoGoMotionLockYjog : Bool;
         NoGoMotionLockZ1move : Bool;
         NoGoMotionLockZ1jog : Bool;
         NoGoMotionLockZ2move : Bool;
         NoGoMotionLockZ2jog : Bool;
         HomingPermissionX : Bool;
         HomingPermissionY : Bool;
         HomingPermissionZ1 : Bool;
         HomingPermissionZ2 : Bool;
         NoGoAlwaysOn : Bool;
      END_STRUCT;
      NoGoZone01Status : Struct   // Status of the NoGoZone with restricted access
         NoGoZone01Active : Bool;
         YouAreInNoGoZone01 : Bool;
         CollisionErrorNoGoZone01 : Bool;
      END_STRUCT;
      PrintingStatus : Struct   // Printing Status Input from NOAH
         InPrintStarted : Bool;   // Input from Noah if the print was started
         InPrintPaused : Bool;   // Input from Noah if the print was paused
         InPrintEnded : Bool;   // Input from Noah if the print was ended
         OutMissingLayerDetected : Bool;   // Missing Layer Detection From The PLC
      END_STRUCT;
   END_VAR
BEGIN
END_DATA_BLOCK

DATA_BLOCK "AXES_Positions_Delays"   // DB33
{ S7_Optimized_Access := 'TRUE' }
VERSION : 0.1
   VAR
      AXIS_X_Position_DelayIn : Bool;
      AXIS_X_Position_DelayOut : Bool;
      AXIS_Y_Position_DelayIn : Bool;
      AXIS_Y_Position_DelayOut : Bool;
      AXIS_Z1_Position_DelayIn : Bool;
      AXIS_Z1_Position_DelayOut : Bool;
      AXIS_Z2_Position_DelayIn : Bool;
      AXIS_Z2_Position_DelayOut : Bool;
   END_VAR
BEGIN
END_DATA_BLOCK

DATA_BLOCK "FTON_FirstTurnON"   // DB46
{ S7_Optimized_Access := 'TRUE' }
VERSION : 0.1
   VAR
      FTON_Enabled_Devices : Bool;
      FTON_Ready_Devices : Bool;
      FTON_IR_Heater_Test : Bool;
      FTON_Door_Sensor_Global : Bool := false;   // Disable Global Sensors
      FTON_Door_Sensor_FS : Bool := false;   // Disable Fluid Supply Sensor
      FTON_Data_Logging_CreateFile : Bool := false;
      FTON_Data_Logging_StartLogging : Bool;
      FTON_Turn_On_Test_Blocks : Bool;
      FTON_Run_Test_01 : Bool;
      FTON_UV_Status_Fake : Bool;
      FTON_ControlButtons : Bool := false;
      FTON_ZAxisDiagnostic : Bool := false;
   END_VAR
BEGIN
END_DATA_BLOCK

DATA_BLOCK "Valuestobelogged"   // DB57
{ S7_Optimized_Access := 'TRUE' }
VERSION : 0.1
   VAR
      Datatobelogged : Struct
         Variable01_Bool : Bool;
         Variable02_Bool : Bool;
         Variable03_Dint : DInt;
         Variable04_Dint : DInt;
         Variable05_Dint : DInt;
         Variable06_Dint : DInt;
      END_STRUCT;
      LogColumns : String := 'Column01, Column02, Column03, Column04, Column05, Column06';
   END_VAR
BEGIN
END_DATA_BLOCK

DATA_BLOCK "CMMS_Z1_FML_REF"   // DB68
{ S7_Optimized_Access := 'TRUE' }
VERSION : 0.1
   VAR
      FML_REF : "DT_FML_REF";
   END_VAR
BEGIN
   FML_REF.DeviceType := 'CMMS';
END_DATA_BLOCK

DATA_BLOCK "CMMS_Z2_FML_REF"   // DB69
{ S7_Optimized_Access := 'TRUE' }
VERSION : 0.1
   VAR
      FML_REF : "DT_FML_REF";
   END_VAR
BEGIN
   FML_REF.DeviceType := 'CMMS';
END_DATA_BLOCK

DATA_BLOCK "Tests_Executing"   // DB97
{ S7_Optimized_Access := 'TRUE' }
VERSION : 0.1
   VAR
      Test01_Enable : Bool;   // Z2 Relative Motion Test Enable
      Test01_Start : Bool;   // Z2 Relative Motion Test Start
      Test01_End : Bool;   // Z2 Relative Motion Test End
   END_VAR
BEGIN
END_DATA_BLOCK

DATA_BLOCK "DB 333"   // DB333
{ S7_Optimized_Access := 'FALSE' }
AUTHOR : AWP_S7P
FAMILY : WEB
VERSION : 1.0
   VAR
      magic : DWord := DW#16#41575043;
      consistency_tag : DWord := DW#16#0F12B01D;
      db_version : Word := W#16#0001;
      length : UInt := 586;
      pagetab_of : UInt := 92;
      pagetab_count : UInt := 4;
      excludetab_of : UInt := 132;
      excludetab_count : UInt := 0;
      fragmentlist_of : UInt := 132;
      fragmentlist_count : UInt := 5;
      fragmenttab_of : UInt := 148;
      fragmenttab_count : UInt := 5;
      datatab_of : UInt := 218;
      datatab_count : UInt := 2;
      usenametab_of : UInt := 226;
      usenametab_count : UInt := 0;
      enumreftab_of : UInt := 226;
      enumreftab_count : UInt := 0;
      enumtab_of : UInt := 226;
      enumtab_count : UInt := 0;
      textlist_of : UInt := 226;
      textlist_count : UInt := 360;
      language_frag_tab_of : UInt := 142;
      language_frag_tab_count : UInt := 6;
      application_name : UInt := 1;
      application_url : UInt := 19;
      application_desc : UInt := 29;
      enum_defs_fragment_start : UInt := 0;
      enum_defs_fragment_count : UInt := 0;
      commandstate : Struct
         last_error : Int := 0;
         debug_mode : Int := 0;
         init : Bool := True;
         deactivate : Bool := False;
         initializing : Bool := False;
         error : Bool := False;
         deactivating : Bool := False;
         deactivated : Bool := False;
         initialized : Bool := False;
         reserved1 : Bool := False;
         reserved2 : Byte := B#16#00;
      END_STRUCT;
      requesttab : Array[1..4] of Struct
         page_index : UInt;
         fragment_index : UInt;
         continue : Bool;
         "repeat" : Bool;
         abort : Bool;
         finish : Bool;
         idle : Bool;
         waiting : Bool;
         sending : Bool;
         aborting : Bool;
         reserved3 : Byte;
      END_STRUCT;
      pagetab : Array[1..4] of Struct
         index : UInt;
         url : UInt;
         mime_type : UInt;
         fragment_start : UInt;
         fragment_num : UInt;
      END_STRUCT;
      fragmentlist : Array[1..5] of UInt;
      language_frag_tab : Struct
         max_language : UInt := 0;
         fragment_count : UInt := 0;
         nolang_offset : UInt := 0;
      END_STRUCT;
      fragmenttab : Array[1..5] of Struct
         fragment_name : UInt;
         fragment_type : Byte;
         fragment_version : Byte;
         content_db : UInt;
         content_of : UInt;
         content_length : UInt;
         data_start : UInt;
         data_num : UInt;
      END_STRUCT;
      datatab : Array[1..2] of Struct
         variable_name : UInt;
         direction : Int;
      END_STRUCT;
      textlist : Array[1..360] of Byte := 434F4E435233444557656253657276657200696E6465782E68746D00434F4E435233444557656253657276657200636F6E63723364655F736F6C6F6C6F676F5F313030783130305F314D335F69636F6E2E69636F006170706C69636174696F6E2F6F637465742D73747265616D00696E6465782E68746D00746578742F68746D6C00494F436F756E7465722E68746D00746578742F68746D6C006A71756572792D322E302E322E6D696E2E6A73006170706C69636174696F6E2F6A61766173637269707400636F6E63723364655F736F6C6F6C6F676F5F313030783130305F314D335F69636F6E2E69636F00696E6465782E68746D00494F436F756E7465722E68746D006A71756572792D322E302E322E6D696E2E6A73006A71756572792D322E302E322E6D696E2E6A735F31002244657654657374426C6F636B222E57656253657276657254657374002244657654657374426C6F636B222E5765625365727665725465737400;
   END_VAR
BEGIN
   requesttab[1..4].page_index := 0;
   requesttab[1..4].fragment_index := 0;
   requesttab[1..4].continue := False;
   requesttab[1..4]."repeat" := False;
   requesttab[1..4].abort := False;
   requesttab[1..4].finish := False;
   requesttab[1..4].idle := False;
   requesttab[1..4].waiting := False;
   requesttab[1..4].sending := False;
   requesttab[1..4].aborting := False;
   requesttab[1..4].reserved3 := B#16#00;
   pagetab[1].index := 1;
   pagetab[2].index := 2;
   pagetab[3].index := 3;
   pagetab[4].index := 4;
   pagetab[1].url := 47;
   pagetab[2].url := 111;
   pagetab[3].url := 131;
   pagetab[4].url := 155;
   pagetab[1].mime_type := 86;
   pagetab[2].mime_type := 121;
   pagetab[3].mime_type := 145;
   pagetab[4].mime_type := 175;
   pagetab[1].fragment_start := 1;
   pagetab[2].fragment_start := 2;
   pagetab[3].fragment_start := 3;
   pagetab[4].fragment_start := 4;
   pagetab[1..3].fragment_num := 1;
   pagetab[4].fragment_num := 2;
   fragmentlist[1] := 1;
   fragmentlist[2] := 2;
   fragmentlist[3] := 3;
   fragmentlist[4] := 4;
   fragmentlist[5] := 5;
   fragmenttab[1].fragment_name := 198;
   fragmenttab[2].fragment_name := 237;
   fragmenttab[3].fragment_name := 247;
   fragmenttab[4].fragment_name := 261;
   fragmenttab[5].fragment_name := 281;
   fragmenttab[1..5].fragment_type := B#16#00;
   fragmenttab[1..5].fragment_version := B#16#00;
   fragmenttab[1..3].content_db := 334;
   fragmenttab[4].content_db := 335;
   fragmenttab[5].content_db := 336;
   fragmenttab[1].content_of := 8;
   fragmenttab[2].content_of := 41248;
   fragmenttab[3].content_of := 42946;
   fragmenttab[4..5].content_of := 8;
   fragmenttab[1].content_length := 41239;
   fragmenttab[2].content_length := 1697;
   fragmenttab[3].content_length := 183;
   fragmenttab[4].content_length := 65526;
   fragmenttab[5].content_length := 17975;
   fragmenttab[1].data_start := 0;
   fragmenttab[2].data_start := 1;
   fragmenttab[3].data_start := 2;
   fragmenttab[4..5].data_start := 0;
   fragmenttab[1].data_num := 0;
   fragmenttab[2..3].data_num := 1;
   fragmenttab[4..5].data_num := 0;
   datatab[1].variable_name := 303;
   datatab[2].variable_name := 332;
   datatab[1..2].direction := 3;
END_DATA_BLOCK

